METHOD PUBLIC OnceEvent
VAR_INPUT
	EventName : T_MaxString;
	EventHandler : I_EventHandler;
END_VAR
eventEmitter.OnceEvent(EventName, EventHandler);
END_METHOD

METHOD PUBLIC OnEvent
VAR_INPUT
	EventName : T_MaxString;
	EventHandler : I_EventHandler;
END_VAR
eventEmitter.OnEvent(EventName, EventHandler);
END_METHOD

METHOD RegisterAsynchronousRpcHandlersWith
VAR_INPUT
	Host : I_HostAsynchronousRpcHandlers;
END_VAR
Host.RegisterHandler('CreateGraph', createGraphRpcHandler);
Host.RegisterHandler('GetStatus', getStatusRpcHandler);
Host.RegisterHandler('GetBlueprints', getBlueprintsRpcHandler);
Host.RegisterHandler('GetContentValue', getContentValueHandler);
Host.RegisterHandler('UpdateParameterValue', updateParameterValueHandler);
END_METHOD

METHOD RegisterSynchronousRpcHandlersWith
VAR_INPUT
	Host : I_HostSynchronousRpcHandlers;
END_VAR
// no implementation
END_METHOD

END_FUNCTION_BLOCK

// Graph/Interfaces/I_HostGraphs
INTERFACE I_HostGraphs

PROPERTY Graphs : I_Graphs
GET
END_GET
END_PROPERTY

END_INTERFACE

// Graph/Host/GraphHost
{attribute 'linkalways'} 
{attribute 'no_explicit_call' := 'This FB is a CLASS and must be accessed using methods or properties'}
{attribute 'enable_dynamic_creation'}
FUNCTION_BLOCK GraphHost IMPLEMENTS I_Graphs, I_Serializable
VAR
	hostParent : I_HostGraphs;
	eventTarget : I_EventTarget;
	graphs : OrderedDictionary;	
END_VAR

METHOD FB_init : BOOL
VAR_INPUT
	bInitRetains : BOOL; // if TRUE, the retain variables are initialized (warm start / cold start)
	bInCopyCode : BOOL;  // if TRUE, the instance afterwards gets moved into the copy code (online change)
	Parent : I_HostGraphs;
	ParentEventTarget : I_EventTarget;
END_VAR
hostParent := Parent;
eventTarget := parentEventTarget;
END_METHOD

METHOD PROTECTED EmitOnGraphAddedEvent
VAR_INPUT
	Graph : I_Graph;
END_VAR
VAR
	graphAddedEvent : GraphAddedEvent(Target := Graph);
END_VAR
IF eventTarget = 0 THEN
	RETURN;
END_IF

eventTarget.Emit('OnGraphAdded', graphAddedEvent);
END_METHOD

METHOD PUBLIC Accept
VAR_INPUT
	visitor : I_GraphVisitor;
END_VAR
VAR
	enumerator : I_ForwardEnumerator;
	graph : I_Graph;
END_VAR
enumerator := graphs.GetEnumerator();

WHILE (enumerator.MoveNext()) DO
	
	IF enumerator.TryGet(graph) THEN
		graph.Accept(Visitor);
	END_IF

END_WHILE

enumerator.Dispose();
END_METHOD

METHOD PUBLIC AddGraph
VAR_INPUT
	Graph : I_Graph;
END_VAR
graphs.AddOrUpdate(Graph.Uuid, Graph);
EmitOnGraphAddedEvent(Graph);
END_METHOD

METHOD PUBLIC DisposeAll
VAR_INPUT
END_VAR
VAR
	enumerator : I_ForwardEnumerator;
	graph : I_Graph;
END_VAR
enumerator := graphs.GetEnumerator();

WHILE enumerator.MoveNext() DO
	IF enumerator.TryGet(graph) THEN
		graph.Dispose();
	END_IF
END_WHILE

graphs.Clear();

enumerator.Dispose();
END_METHOD

METHOD PUBLIC Execute
VAR_INPUT
END_VAR
VAR
	enumerator : I_ForwardEnumerator;
	graph : I_Graph;
END_VAR
enumerator := graphs.GetEnumerator();

WHILE enumerator.MoveNext() DO
	IF enumerator.TryGet(graph) THEN
		graph.Execute();
	END_IF
END_WHILE

enumerator.Dispose();
END_METHOD

METHOD PUBLIC RemoveGraph
VAR_INPUT
	Graph : I_Graph;
END_VAR
graphs.Remove(Graph.Uuid);
END_METHOD

METHOD PUBLIC SerializeWith
VAR_INPUT
	Serializer : I_Serializer;
END_VAR
VAR
	enumerator : I_ForwardEnumerator;
	graph : I_Graph;
END_VAR
IF graphs.Count = 0 THEN
	RETURN;
END_IF

Serializer.AddKey('graphs');
Serializer.StartArray();

enumerator := graphs.GetEnumerator();

WHILE enumerator.MoveNext() DO
	IF enumerator.TryGet(graph) THEN
		graph.SerializeWith(Serializer);
	END_IF
END_WHILE

Serializer.EndArray();
enumerator.Dispose();
END_METHOD

METHOD PUBLIC TryGetGraphByUuid : BOOL
VAR_INPUT
	Uuid : T_MAXSTRING;
	Destination : REFERENCE TO I_Graph;
END_VAR
VAR
	graph : I_Graph;
END_VAR
IF NOT graphs.TryGetValue(Uuid, graph) THEN
	RETURN;
END_IF

Destination := graph;
TryGetGraphByUuid := TRUE;
END_METHOD

END_FUNCTION_BLOCK

// Graph/Events/GraphAddedEvent
{attribute 'linkalways'} 
{attribute 'no_explicit_call' := 'This FB is a CLASS and must be accessed using methods or properties'}
{attribute 'enable_dynamic_creation'}
FUNCTION_BLOCK GraphAddedEvent EXTENDS Disposable IMPLEMENTS I_GraphAddedEvent
VAR
	_target : I_Graph;
END_VAR

METHOD FB_init : BOOL
VAR_INPUT
	bInitRetains : BOOL; // if TRUE, the retain variables are initialized (warm start / cold start)
	bInCopyCode : BOOL;  // if TRUE, the instance afterwards gets moved into the copy code (online change)
	Target : I_Graph;
END_VAR
THIS^._target := Target;
END_METHOD

PROPERTY PUBLIC Target : I_Graph
GET
Target := _target;
END_GET
END_PROPERTY

END_FUNCTION_BLOCK

// Graph/Events/I_GraphAddedEvent
INTERFACE I_GraphAddedEvent EXTENDS I_Event

PROPERTY PUBLIC Target : I_Graph
GET
END_GET
END_PROPERTY

END_INTERFACE

// Extensions/Namespace/ExtensionNamespace
{attribute 'linkalways'} 
{attribute 'no_explicit_call' := 'This FB is a CLASS and must be accessed using methods or properties'}
{attribute 'enable_dynamic_creation'}
FUNCTION_BLOCK ExtensionNamespace
VAR
	_extensionName : T_MAXSTRING;
	_targetName : T_MAXSTRING;
	_isExtensionPath : BOOL;
END_VAR

METHOD FB_init : BOOL
VAR_INPUT
	bInitRetains : BOOL; // if TRUE, the retain variables are initialized (warm start / cold start)
	bInCopyCode : BOOL;  // if TRUE, the instance afterwards gets moved into the copy code (online change)
	Path : T_MAXSTRING;
END_VAR
Initialize(Path);
END_METHOD

PROPERTY PUBLIC ExtensionName : T_MAXSTRING
GET
IF NOT _isExtensionPath THEN
	RETURN;
END_IF

ExtensionName := _extensionNAme;
END_GET
END_PROPERTY

METHOD PUBLIC Initialize
VAR_INPUT
	Path : T_MAXSTRING;
END_VAR
_isExtensionPath := FindAndSplitChar(
	sSeparatorChar := '.',  
	pSrcString := ADR(Path),                                  
	pLeftString := ADR(_extensionName),   
	nLeftSize := SIZEOF(_extensionName),                                  
	pRightString := ADR(_targetName), 
	nRightSize := SIZEOF(_targetName),                                
	bSearchFromRight := TRUE 
);
END_METHOD

PROPERTY PUBLIC IsExtensionPath : BOOL
GET
IsExtensionPath := _isExtensionPath;
END_GET
END_PROPERTY

PROPERTY PUBLIC TargetName : T_MAXSTRING
GET
IF NOT _isExtensionPath THEN
	RETURN;
END_IF

TargetName := _targetName;
END_GET
END_PROPERTY

END_FUNCTION_BLOCK

// Extensions/PreExecutionCheck/Alarms/PreExecutionCheckFailedAlarm
{attribute 'linkalways'} 
{attribute 'no_explicit_call' := 'This FB is a CLASS and must be accessed using methods or properties'}
{attribute 'enable_dynamic_creation'}
FUNCTION_BLOCK PUBLIC PreExecutionCheckFailedAlarm EXTENDS Alarm
VAR
	state : (CLEARED, RAISED);
	_reason : T_MAXSTRING;
END_VAR

PROPERTY Active : BOOL
GET
Active := state <> CLEARED;
END_GET
END_PROPERTY

METHOD PUBLIC Clear
_reason := '';
state := CLEARED;
END_METHOD

PROPERTY PUBLIC Message : T_MaxString
GET
Message := 'Pre-execution check failed';
END_GET
END_PROPERTY

METHOD PUBLIC Raise
VAR_INPUT
	Reason : T_MAXSTRING;
END_VAR
_reason := Reason;
state := RAISED;
END_METHOD

PROPERTY Reason : T_MaxString
GET
Reason := _reason;
END_GET
END_PROPERTY

END_FUNCTION_BLOCK

// Extensions/PreExecutionCheck/Checks/I_PreExecutionChecks
INTERFACE I_PreExecutionChecks

METHOD PUBLIC Fail
VAR_INPUT
	Message : T_MAXSTRING;
END_VAR
END_METHOD

PROPERTY PUBLIC Failed : BOOL
GET
END_GET
END_PROPERTY

METHOD PUBLIC IsFalse
VAR_INPUT
	Actual : BOOL;
	Message : T_MAXSTRING;
END_VAR
END_METHOD

METHOD PUBLIC IsTrue
VAR_INPUT
	Actual : BOOL;
	Message : T_MAXSTRING;
END_VAR
END_METHOD

END_INTERFACE

// Extensions/PreExecutionCheck/Checks/PreExecutionChecks
FUNCTION_BLOCK PreExecutionChecks IMPLEMENTS I_PreExecutionChecks
VAR
	hasFailed : BOOL;
	hasFailedReason : T_MAXSTRING;
END_VAR;

METHOD PUBLIC Fail
VAR_INPUT
	Message : T_MAXSTRING;
END_VAR
IF hasFailed THEN
	RETURN;
END_IF

hasFailed := TRUE;
hasFailedReason := Message;
END_METHOD

PROPERTY PUBLIC Failed : BOOL
GET
Failed := hasFailed;
END_GET
END_PROPERTY

METHOD PUBLIC IsFalse
VAR_INPUT
	Actual : BOOL;
	Message : T_MAXSTRING;
END_VAR
IF hasFailed THEN
	RETURN;
END_IF

IF NOT Actual THEN
	RETURN;
END_IF

hasFailed := TRUE;
hasFailedReason := Message;
END_METHOD

METHOD PUBLIC IsTrue
VAR_INPUT
	Actual : BOOL;
	Message : T_MAXSTRING;
END_VAR
IF hasFailed THEN
	RETURN;
END_IF

IF Actual THEN
	RETURN;
END_IF

hasFailed := TRUE;
hasFailedReason := Message;
END_METHOD

PROPERTY PUBLIC Passed : BOOL
GET
Passed := not hasFailed;
END_GET
END_PROPERTY

PROPERTY PUBLIC Reason : T_MAXSTRING
GET
Reason := hasFailedReason;
END_GET
END_PROPERTY

METHOD PUBLIC Reset
VAR_INPUT
END_VAR
hasFailed := FALSE;
hasFailedReason := '';
END_METHOD

END_FUNCTION_BLOCK

// Extensions/PreExecutionCheck/Interfaces/I_PreCheckedNode
INTERFACE I_PreCheckedNode EXTENDS I_Node

METHOD PreExecutionCheck
VAR_INPUT
	Check : I_PreExecutionChecks;
END_VAR
END_METHOD

END_INTERFACE

// Extensions/PreExecutionCheck/PreExecutionCheckExtension
FUNCTION_BLOCK PreExecutionCheckExtension EXTENDS Extension IMPLEMENTS I_EventHandler
VAR
	parentAsPreCheckedNode : I_PreCheckedNode;
	preExecutionCheckFailedAlarm : PreExecutionCheckFailedAlarm(THIS^);
	enable : _BOOL(TRUE);
END_VAR

METHOD FB_init : BOOL
VAR_INPUT
	bInitRetains : BOOL; // if TRUE, the retain variables are initialized (warm start / cold start)
	bInCopyCode : BOOL;  // if TRUE, the instance afterwards gets moved into the copy code (online change)
	Name : T_MAXSTRING;
	Parent : I_HostExtensions;
END_VAR
AddParameter('enable', enable);

IF NOT __QUERYINTERFACE(Parent, parentAsPreCheckedNode) THEN
	RETURN;
END_IF

RegisterForPreExecuteEvent();
END_METHOD

METHOD FB_exit : BOOL
VAR_INPUT
	bInCopyCode : BOOL; // if TRUE, the exit method is called for exiting an instance that is copied afterwards (online change).
END_VAR
IF bInCopyCode THEN
	RETURN;
END_IF

DeregisterForPreExecuteEvent();
END_METHOD

METHOD PRIVATE DeregisterForPreExecuteEvent
VAR_INPUT
END_VAR
IF parentAsPreCheckedNode = 0 THEN
	RETURN;
END_IF

parentAsPreCheckedNode.OffEvent('OnNodePreExecute', THIS^);
END_METHOD

METHOD PRIVATE RegisterForPreExecuteEvent
VAR_INPUT
END_VAR
IF parentAsPreCheckedNode = 0 THEN
	RETURN;
END_IF

parentAsPreCheckedNode.OnEvent('OnNodePreExecute', THIS^);
END_METHOD

METHOD PUBLIC HandleEvent
VAR_INPUT
	Event : I_Event;
END_VAR
VAR
	nodePreExecuteEvent : I_NodePreExecuteEvent;
	preExecutionChecks : PreExecutionChecks;
END_VAR
IF NOT enable.Value THEN
	IF preExecutionCheckFailedAlarm.Active THEN
		preExecutionCheckFailedAlarm.Clear();
	END_IF
	RETURN;
END_IF

IF NOT __QUERYINTERFACE(Event, nodePreExecuteEvent) THEN
	RETURN;
END_IF

parentAsPreCheckedNode.PreExecutionCheck(preExecutionChecks);
IF preExecutionChecks.Failed THEN
	preExecutionCheckFailedAlarm.Raise(preExecutionChecks.Reason);
	nodePreExecuteEvent.Cancel();
	RETURN;
END_IF

preExecutionCheckFailedAlarm.Clear();
END_METHOD

END_FUNCTION_BLOCK

// IecDatatypesPack/IecDatatypesPack
{attribute 'linkalways'} 
{attribute 'no_explicit_call' := 'This FB is a CLASS and must be accessed using methods or properties'}
{attribute 'enable_dynamic_creation'}
FUNCTION_BLOCK IecDatatypesPack IMPLEMENTS I_GraphPack
VAR
	// _bit not included as this can only be part of a structure
	_bool : _BOOL(FALSE);
	_byte : _BYTE(0);
	_dint : _DINT(0);
	_dt : _DT(DT#1970-1-1-0:0:0);
	_dword : _DWORD(0);
	_int : _INT(0);
	_lint : _LINT(0);
	_lreal : _LREAL(0);
	_lword : _LWORD(0);
	_real : _REAL(0);
	_sint : _SINT(0);
	_time_of_day : _TIME_OF_DAY(TOD#0:0:0);
	_tod : _TOD(TOD#0:0:0);
	_udint : _UDINT(0);
	_uint : _UINT(0);
	_ulint : _ULINT(0);
	_usint : _USINT(0);
	_word : _WORD(0);
    _string : _STRING('');
	_pvoid : _PVOID;
END_VAR

METHOD RegisterWithDatatypes
VAR_INPUT
	Datatypes : I_Datatypes;
END_VAR
Datatypes.RegisterDatatype(_bool);
Datatypes.RegisterDatatype(_byte);
Datatypes.RegisterDatatype(_dint);
Datatypes.RegisterDatatype(_dt);
Datatypes.RegisterDatatype(_dword);
Datatypes.RegisterDatatype(_int);
Datatypes.RegisterDatatype(_lint);
Datatypes.RegisterDatatype(_lreal);
Datatypes.RegisterDatatype(_lword);
Datatypes.RegisterDatatype(_real);
Datatypes.RegisterDatatype(_sint);
Datatypes.RegisterDatatype(_time_of_day);
Datatypes.RegisterDatatype(_tod);
Datatypes.RegisterDatatype(_udint);
Datatypes.RegisterDatatype(_uint);
Datatypes.RegisterDatatype(_ulint);
Datatypes.RegisterDatatype(_usint);
Datatypes.RegisterDatatype(_word);
Datatypes.RegisterDatatype(_string);
Datatypes.RegisterDatatype(_pvoid);
END_METHOD

METHOD PUBLIC RegisterWithNodeFactory
VAR_INPUT
	NodeFactory : I_NodeFactory;
END_VAR
// not implemented
END_METHOD

END_FUNCTION_BLOCK

// Node/Hardware/HardwareNode
{attribute 'linkalways'} 
{attribute 'no_explicit_call' := 'This FB is a CLASS and must be accessed using methods or properties'}
{attribute 'enable_dynamic_creation'}
{attribute 'hide_all_locals'}
FUNCTION_BLOCK ABSTRACT HardwareNode EXTENDS Node
VAR
END_VAR

METHOD PUBLIC  Clone : I_Node
VAR_INPUT
END_VAR
Clone := THIS^;
// hardware nodes are singletons, so when asked to clone, it instead returns itself.
END_METHOD

METHOD PUBLIC Dispose
VAR_INPUT
END_VAR
// hardware nodes are singletons, so this remains empty as it should not be destroyed.
END_METHOD

END_FUNCTION_BLOCK
